Staubli VAL3: onStart.pgx

program onStart()
  local num i
  local string l_sPath
  local string l_sMessage
begin
  // logMsg
  logMsg("[KERNEL] INTERFACE:PAGE PALLET")
  // reset the exit button
  bExit=false
  // reset the Key pressure
  call use:nullKey(nKey)
  nIndex=0
  // load the TRAJ
  sPalletName=sItems
  // define the list
  call pallet:load(sPalletName,i)
  if i!=0
    call language:message(l_sMessage,-7)
    popUpMsg(l_sMessage+"#"+saveData:sTrajTypeUsing+"/"+sPalletName+" ; "+toString("",i))
  endIf
  //
  call buildList()
  // build the page
  call refreshStatic()
  // define the list
end
